ABB RobotStudio station: PROYECTO_BUENO_ROBOTICA.rspag

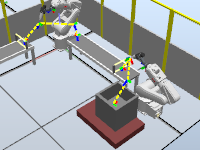
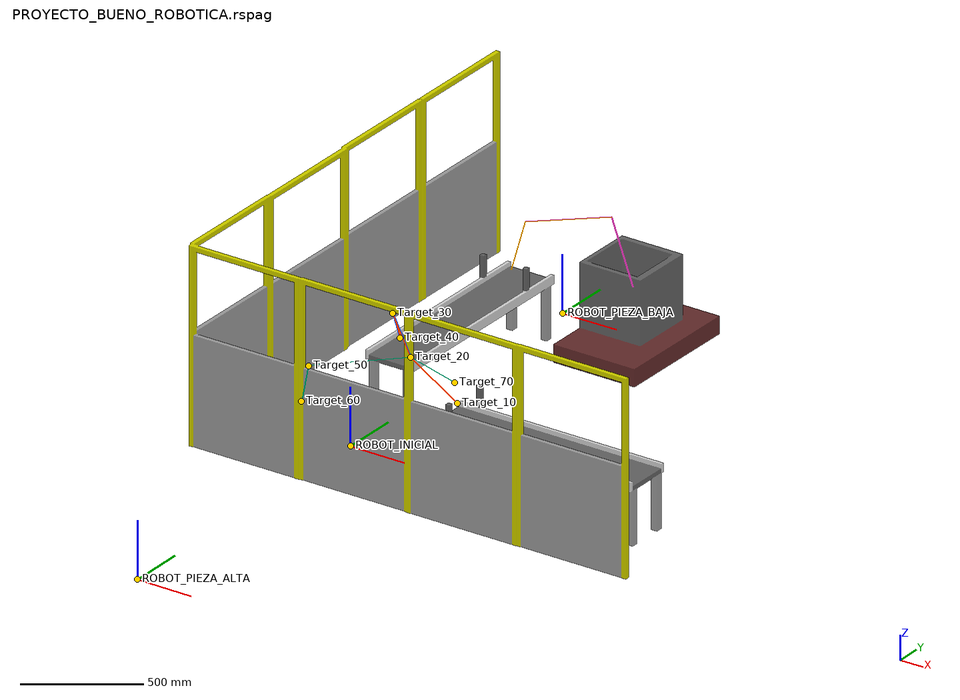
[picture v1: parts stored in the station drawn from their meshes, with robot base, taught points and paths (robot models come from the ABB library and are not in the file)]
--- station ---
Station Station (saved by RobotStudio 21.2.9526.0)
Controller Controlador3, task T_ROB1: task frame (RAPID world) sits at (0, 1493.87, 0) mm, rotated rx 0 ry 0 rz -90 deg in the station
Controller Controlador2, task T_ROB1: task frame (RAPID world) sits at (0, -1501.35, 0) mm, rotated rx 0 ry 0 rz 90 deg in the station
Controller Controlador1
  mechanical unit ROB_1: ROBOT_INICIAL, 6 joints, base frame (0, 0, 0) mm
Controller Controlador2
  mechanical unit ROB_1: ROBOT_PIEZA_ALTA, 6 joints, base frame (0, 0, 0) mm
Controller Controlador3
  mechanical unit ROB_1: ROBOT_PIEZA_BAJA, 6 joints, base frame (0, 0, 0) mm
Layout (positions relative to the parent item):
  - ROBOT_INICIAL [mechanism, from Robots\IRB120_3_58_G_01.rslib] at (0, 0, 0) mm; joint values [0.0153, -0.9412, 0.5438, -0.013, 0.8103, 0.021] (rad or m)
  - CINTA_INICIAL [part] at (1649.16, 0.65, 0) mm, rotated rx 0 ry 0 rz 180 deg, size 1004.2 x 233.8 x 295.1 mm
  - CINTA_PIEZA_BAJA [part] at (-5.09, 92.92, 0) mm, rotated rx 0 ry 0 rz 90 deg, size 1004.2 x 233.8 x 295.1 mm
  - ROBOT_PIEZA_BAJA [mechanism, from Robots\IRB120_3_58_G_01.rslib] at (0, 1493.87, 0) mm, rotated rx 0 ry 0 rz -90 deg; joint values [0, -1.3872, 0.8613, 0, 0.5297, 0] (rad or m)
  - ROBOT_PIEZA_ALTA [mechanism, from Robots\IRB120_3_58_G_01.rslib] at (0, -1501.35, 0) mm, rotated rx 0 ry 0 rz 90 deg; joint values [0, 0, 0, 0, 0.5236, 0] (rad or m)
  - PALE [part] at (-690.19, -1706.89, 0) mm
  - PALE_2 [part] at (226.17, 1105.11, 0) mm, size 400 x 600 x 80 mm
  - PALE_3 [part] at (-668.39, 1113.38, 0) mm
  - PALE_4 [part] at (309.1, -1704.29, 0) mm
  - MyTool [mechanism, from Training Objects\myTool.rslib] at (99.08, 0.84, 601.52) mm, rotated rx 178.96 ry 66.34 rz 179.16 deg
  - MyTool_3 [mechanism, from Training Objects\myTool.rslib] at (0, 1461.27, 551.16) mm, rotated rx 180 ry 89.78 rz 90 deg
  - PROTECCION_7 [part] at (1838.39, -653.58, 0) mm, rotated rx 0 ry 0 rz 90 deg, size 22.3 x 539.4 x 900 mm
  - PROTECCION_8 [part] at (-248.35, 2040.22, 0) mm, rotated rx 0 ry 0 rz 180 deg, size 22.3 x 539.4 x 900 mm
  - SENSOR [part] at (550.47, 98.45, 290.03) mm, size 20 x 20 x 100 mm
  - SENSOR_3 [part] at (31.03, 1015.51, 0) mm
  - SENSOR_4 [part] at (31.03, 1015.51, 0) mm
  - SENSOR_5 [part] at (31.03, 1015.51, 0) mm
  - CINTA_PIEZA_ALTA [part] at (-8.5, -1442.97, 0) mm, rotated rx 0 ry 0 rz 90 deg
  - SENSOR_6 [part] at (-130.12, -1151.13, 289.91) mm
  - SENSOR_7 [part] at (552.16, -120.97, 291.11) mm, size 20 x 20 x 100 mm
  - LineSensor_CINTA_INICIAL_ALTO [smart component, from Components\LineSensor.rslib]
      properties: Start=[0.562162 -0.10097 0.391108]; End=[0.560466 0.098451 0.39003]; Radius=0; SensedPart=SENSOR_7; SensedPoint=[0.562161987304687 -0.100970001220703 0.391108001708984]
    - _sensorPart_ [part], size 1.7 x 199.4 x 1.1 mm
  - LineSensor_CINTA_INICIAL_BAJO [smart component, from Components\LineSensor.rslib]
      properties: Start=[0.560466 0.098451 0.29003]; End=[0.562162 -0.10097 0.291108]; Radius=0; SensedPart=(none); SensedPoint=[0 0 0]
    - _sensorPart_ [part], size 1.7 x 199.4 x 1.1 mm
  - PhysicsControl [smart component, from Components\PhysicsControl.rslib]
      properties: Object=CINTA_INICIAL; Behavior=1; SurfaceVelocity=0.2
  - PhysicsControl_2 [smart component, from Components\PhysicsControl.rslib]
      properties: Object=CINTA_PIEZA_BAJA; Behavior=1; SurfaceVelocity=0.2
  - Attacher [smart component, from Components\Attacher.rslib]
      properties: Parent=MyTool; Flange=0; Child=(none); Mount=false; Offset=[0 0 0]; Orientation=[0 0 0]
  - Detacher [smart component, from Components\Detacher.rslib]
      properties: Child=(none); KeepPosition=true
  - SENSOR_8 [part] at (87, 1086.5, 290.62) mm, size 20 x 20 x 100 mm
  - SENSOR_9 [part] at (-126.77, 1089.55, 289.95) mm, size 20 x 20 x 100 mm
  - SENSOR_10 [part] at (89.27, -1145.05, 289.5) mm
  - LineSensor_CINTA:PIEZA_BAJA_ALTO [smart component, from Components\LineSensor.rslib]
      properties: Start=[0.085996 1.096498 0.390618]; End=[-0.099773 1.099547 0.389951]; Radius=0; SensedPart=(none); SensedPoint=[0 0 0]
    - _sensorPart_ [part], size 185.8 x 3 x 0.7 mm
  - LineSensor_CINTA_PIEZA_BAJA_BAJO [smart component, from Components\LineSensor.rslib]
      properties: Start=[0.076996 1.096498 0.290618]; End=[-0.098773 1.099547 0.289951]; Radius=0; SensedPart=(none); SensedPoint=[0 0 0]
    - _sensorPart_ [part], size 175.8 x 3 x 0.7 mm
  - CAJA [part] at (1364.14, -37.71, 266.99) mm, size 60 x 60 x 60 mm
  - Source [smart component, from Components\Source.rslib]
      properties: Source=CAJA; Copy=(none); Parent=(none); Position=[1.348944 -0.035764 0.27]; Orientation=[0 0 0]; Transient=true; PhysicsBehavior=3
  - Attacher_2 [smart component, from Components\Attacher.rslib]
      properties: Parent=MyTool_3; Flange=0; Child=(none); Mount=false; Offset=[0 0 0]; Orientation=[0 0 0]
  - Detacher_2 [smart component, from Components\Detacher.rslib]
      properties: Child=(none); KeepPosition=true
  - CAJA_GRANDE [part] at (1304.51, -24.93, 274) mm, size 100 x 100 x 150 mm
  - CAJA_GUARDAR [part] at (-496.56, 737.11, 75.2) mm, size 304.8 x 304.8 x 304.8 mm
  - PROTECCION_9 [part] at (225.18, -657.22, 0) mm, rotated rx 0 ry 0 rz 90 deg, size 22.3 x 539.4 x 900 mm
  - PROTECCION_10 [part] at (-242.45, 415.11, 0) mm, rotated rx 0 ry 0 rz 180 deg, size 22.3 x 539.4 x 900 mm
  - PROTECCION_11 [part] at (-239.98, 952.89, 0) mm, rotated rx 0 ry 0 rz 180 deg, size 22.3 x 539.4 x 900 mm
  - PROTECCION_12 [part] at (-248.62, 1492.56, 0) mm, rotated rx 0 ry 0 rz 180 deg, size 22.3 x 539.4 x 900 mm
  - PROTECCION_13 [part] at (764.68, -653.95, 0) mm, rotated rx 0 ry 0 rz 90 deg, size 22.3 x 539.4 x 900 mm
  - PROTECCION_14 [part] at (1298.16, -656.54, 0) mm, rotated rx 0 ry 0 rz 90 deg, size 22.3 x 539.4 x 900 mm
  - Sink [smart component, from Components\Sink.rslib]
      properties: Object=(none)
Attachment: MyTool is attached to ROBOT_INICIAL / Link6
Attachment: MyTool_3 is attached to ROBOT_PIEZA_BAJA / Link6
Station signals: DI CAJA
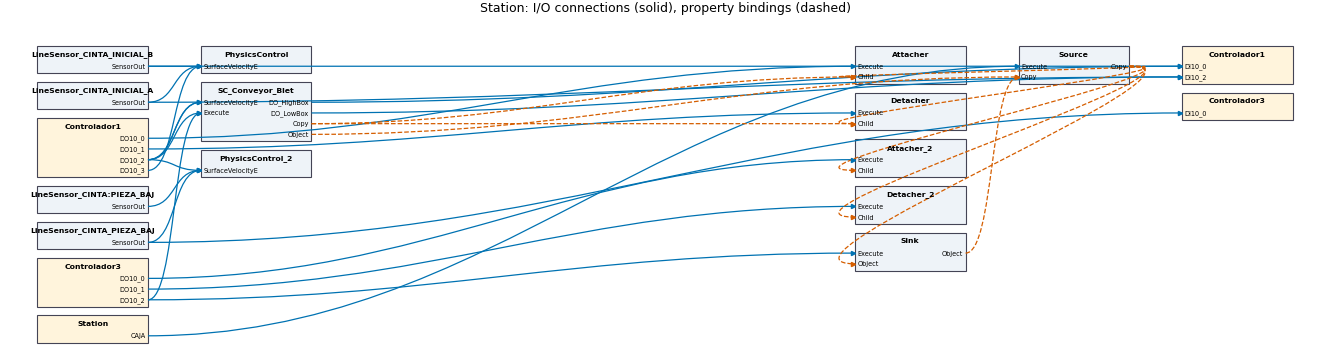
Station logic (signal -> signal, property => property):
  SC_Conveyor_Blet.DO_HighBox -> Controlador1.DI10_0
  SC_Conveyor_Blet.DO_LowBox -> Controlador1.DI10_2
  LineSensor_CINTA_INICIAL_BAJO.SensorOut -> PhysicsControl.SurfaceVelocityEnabled
  LineSensor_CINTA_INICIAL_ALTO.SensorOut -> PhysicsControl.SurfaceVelocityEnabled
  Controlador1.DO10_0 -> Attacher.Execute
  LineSensor_CINTA_INICIAL_BAJO.SensorOut -> Controlador1.DI10_0
  LineSensor_CINTA_INICIAL_ALTO.SensorOut -> Controlador1.DI10_2
  Controlador1.DO10_1 -> Detacher.Execute
  LineSensor_CINTA:PIEZA_BAJA_ALTO.SensorOut -> PhysicsControl_2.SurfaceVelocityEnabled
  LineSensor_CINTA_PIEZA_BAJA_BAJO.SensorOut -> PhysicsControl_2.SurfaceVelocityEnabled
  Controlador1.DO10_2 -> PhysicsControl_3.SurfaceVelocityEnabled
  Controlador1.DO10_3 -> PhysicsControl.SurfaceVelocityEnabled
  Controlador1.DO10_2 -> PhysicsControl_5.SurfaceVelocityEnabled
  Controlador1.DO10_2 -> Source.Execute
  Controlador1.DO10_2 -> PhysicsControl_2.SurfaceVelocityEnabled
  LineSensor_CINTA_PIEZA_BAJA_BAJO.SensorOut -> Controlador3.DI10_0
  Controlador3.DO10_0 -> Attacher_2.Execute
  Controlador3.DO10_1 -> Detacher_2.Execute
  Controlador3.DO10_2 -> Sink.Execute
  Controlador3.DO10_2 -> Sink.Execute
  Station.CAJA -> Source.Execute
  Source.Copy => Attacher.Child
  Source.Copy => Detacher.Child
  Source.Copy => Attacher.Child
  Source.Copy => Detacher.Child
  Source.Copy => Attacher_2.Child
  Source.Copy => Detacher_2.Child
  Sink.Object => Source.Copy
  Sink.Object => Source.Copy
  Source.Copy => Sink.Object

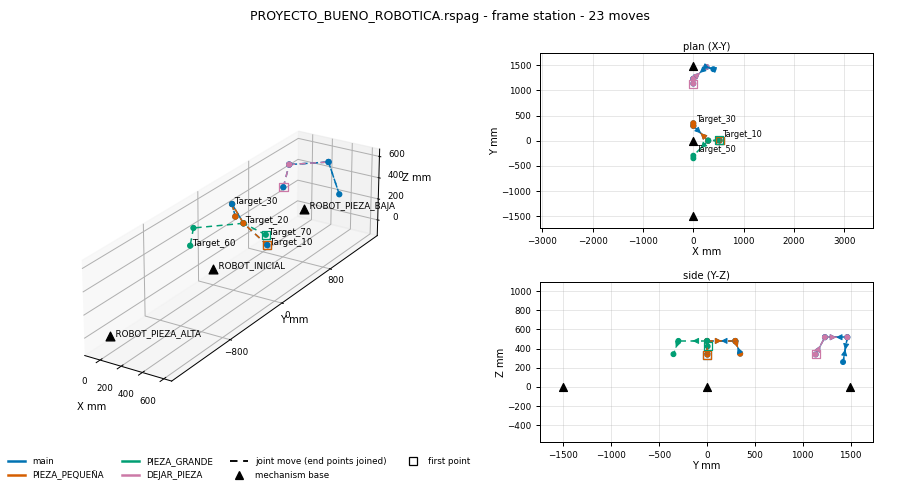
[picture p0: tool path of PROYECTO_BUENO_ROBOTICA.rspag in frame station, 23 of 23 moves have a stored position in this frame; points joined in program order, loops and branches not executed]
--- Backups/Controlador1/RAPID/TASK1/PROGMOD/CalibData.mod ---
MODULE CalibData
    PERS tooldata MyTool:=[TRUE,[[31.7926,0,229.639],[0.945519,0,0.325568,0]],[1,[0,0,1],[1,0,0,0],0,0,0]];
    TASK PERS wobjdata CINTA_1:=[FALSE,TRUE,"",[[0,0,0],[1,0,0,0]],[[0,0,0],[1,0,0,0]]];
ENDMODULE

--- Backups/Controlador1/RAPID/TASK1/PROGMOD/Module1.mod ---
MODULE Module1
        CONST robtarget Target_10:=[[524.488,5.564,337.068],[0.000000001,-0.000000001,1,0],[0,0,0,0],[9E+09,9E+09,9E+09,9E+09,9E+09,9E+09]];
    CONST robtarget Target_20:=[[296.669421919,2.08003687,480.265402411],[0.244840724,-0.000000001,0.969556084,0.003744278],[0,-1,0,0],[9E+09,9E+09,9E+09,9E+09,9E+09,9E+09]];
    CONST robtarget Target_30:=[[0.854294307,296.675483713,480.265402411],[0.171348121,-0.682180871,0.688961725,0.174930904],[1,-1,0,0],[9E+09,9E+09,9E+09,9E+09,9E+09,9E+09]];
    CONST robtarget Target_40:=[[0.578072629,347.819693408,346.913289479],[0.030324355,-0.70294026,0.709927462,0.03095842],[1,-1,0,0],[9E+09,9E+09,9E+09,9E+09,9E+09,9E+09]];
    CONST robtarget Target_50:=[[0.892731255,-296.675394938,480.265369004],[0.175434591,0.686950192,0.684206456,-0.170832265],[-1,-1,0,0],[9E+09,9E+09,9E+09,9E+09,9E+09,9E+09]];
    CONST robtarget Target_60:=[[1.479554637,-348.653016996,341.544953495],[0.025529615,0.708070337,0.705242245,-0.024859873],[-1,-1,0,0],[9E+09,9E+09,9E+09,9E+09,9E+09,9E+09]];
    CONST robtarget Target_70:=[[507.935,8.772,423.995],[0.000000001,-0.000000001,1,0],[0,0,0,0],[9E+09,9E+09,9E+09,9E+09,9E+09,9E+09]];
!***********************************************************
    !
    ! Módulo:  Module1
    !
    ! Descripción:
    !   <Introduzca la descripción aquí>
    !
    ! Autor: javie
    !
    ! Versión: 1.0
    !
    !***********************************************************


    !***********************************************************
    !
    ! Procedimiento Main
    !
    !   Este es el punto de entrada de su programa
    !
    !***********************************************************
    PROC main()
        Set DO10_4;
        Reset DO10_4;
        Set DO10_3;
        Reset DO10_1;
        Reset DO10_0;
        WaitDI DI10_0,1;
        WaitTime 1;
        MoveJ Target_10,v1000,fine,MyTool\WObj:=CINTA_1;
        Set DO10_0;
        WaitTime 1;
        MoveJ Target_20,v1000,fine,MyTool\WObj:=CINTA_1;
        Set DO10_4;
        MoveJ Target_30,v1000,z100,MyTool\WObj:=CINTA_1;
        MoveJ Target_40,v1000,fine,MyTool\WObj:=CINTA_1;
        Set DO10_1;
        Set DO10_2;
        WaitTime 1;
        MoveJ Target_30,v1000,z100,MyTool\WObj:=CINTA_1;
        MoveJ Target_20,v1000,fine,MyTool\WObj:=CINTA_1;


    ENDPROC
    PROC PIEZA_PEQUEÑA()
        MoveJ Target_10,v1000,fine,MyTool\WObj:=CINTA_1;
        MoveJ Target_20,v1000,fine,MyTool\WObj:=CINTA_1;
        MoveJ Target_30,v1000,z100,MyTool\WObj:=CINTA_1;
        MoveJ Target_40,v1000,fine,MyTool\WObj:=CINTA_1;
    ENDPROC
    PROC PIEZA_GRANDE()
        MoveJ Target_70,v200,fine,MyTool\WObj:=CINTA_1;
        MoveJ Target_20,v1000,fine,MyTool\WObj:=CINTA_1;
        MoveJ Target_50,v1000,fine,MyTool\WObj:=CINTA_1;
        MoveJ Target_60,v1000,fine,MyTool\WObj:=CINTA_1;
    ENDPROC
ENDMODULE

--- Backups/Controlador2/RAPID/TASK1/PROGMOD/Module1.mod ---
MODULE Module1
    !***********************************************************
    !
    ! Módulo:  Module1
    !
    ! Descripción:
    !   <Introduzca la descripción aquí>
    !
    ! Autor: javie
    !
    ! Versión: 1.0
    !
    !***********************************************************


    !***********************************************************
    !
    ! Procedimiento Main
    !
    !   Este es el punto de entrada de su programa
    !
    !***********************************************************
    PROC main()
        !Añada aquí su código
    ENDPROC
ENDMODULE

--- Backups/Controlador3/RAPID/TASK1/PROGMOD/CalibData.mod ---
MODULE CalibData
    PERS tooldata MyTool:=[TRUE,[[31.792631019,0,229.638935148],[0.945518576,0,0.325568154,0]],[1,[0,0,1],[1,0,0,0],0,0,0]];
ENDMODULE

--- Backups/Controlador3/RAPID/TASK1/PROGMOD/Module1.mod ---
MODULE Module1
        CONST robtarget Target_10:=[[358.458066847,0,338.786730568],[0.146240119,0,0.989249123,0],[0,0,0,0],[9E+09,9E+09,9E+09,9E+09,9E+09,9E+09]];
    CONST robtarget Target_20:=[[262.109517355,0,518.483225276],[0.43664348,0,0.899634632,0],[0,0,0,4],[9E+09,9E+09,9E+09,9E+09,9E+09,9E+09]];
    CONST robtarget Target_30:=[[28.317745802,260.57533337,518.483225276],[0.325004428,-0.600792335,0.669620072,0.291598441],[0,0,-1,4],[9E+09,9E+09,9E+09,9E+09,9E+09,9E+09]];
    CONST robtarget Target_40:=[[72.897632969,399.258136435,259.476555382],[0.009818398,-0.640410998,0.767925978,0.008188042],[0,0,-1,0],[9E+09,9E+09,9E+09,9E+09,9E+09,9E+09]];
    CONST robtarget Target_50:=[[124.528656109,351.162,140.028],[0,-0.707106781,0.707106782,0],[0,0,0,0],[9E+09,9E+09,9E+09,9E+09,9E+09,9E+09]];

!***********************************************************
    !
    ! Módulo:  Module1
    !
    ! Descripción:
    !   <Introduzca la descripción aquí>
    !
    ! Autor: javie
    !
    ! Versión: 1.0
    !
    !***********************************************************


    !***********************************************************
    !
    ! Procedimiento Main
    !
    !   Este es el punto de entrada de su programa
    !
    !***********************************************************
    PROC main()

       Reset DO10_0;
       Reset DO10_1;
       Reset DO10_2;
       WaitDI DI10_0,1;
       MoveJ Target_10,v200,fine,MyTool\WObj:=wobj0;
       WaitTime 1;
       Set DO10_0;
       WaitTime 0.5;
       MoveJ Target_20,v200,fine,MyTool\WObj:=wobj0;
       MoveJ Target_30,v200,fine,MyTool\WObj:=wobj0;
       MoveJ Target_40,v1000,z100,MyTool\WObj:=wobj0;
       Waittime 1;
       Set DO10_1;
       Set DO10_2;
       MoveJ Target_30,v200,fine,MyTool\WObj:=wobj0;
       MoveJ Target_20,v200,fine,MyTool\WObj:=wobj0;
       Set DO10_3;

    ENDPROC
    PROC DEJAR_PIEZA()
        MoveJ Target_10,v200,fine,MyTool\WObj:=wobj0;
        MoveJ Target_20,v1000,fine,MyTool\WObj:=wobj0;
        MoveJ Target_30,v1000,fine,MyTool\WObj:=wobj0;




    ENDPROC
ENDMODULE

--- Backups/Controlador1/SYSPAR/EIO.cfg ---
EIO:CFG_1.0:6:1::
#
INDUSTRIAL_NETWORK:

      -Name "DeviceNet" -Label "DeviceNet Master/Slave Network" -Address "2"
#
DEVICENET_DEVICE:

      -Name "d652" -VendorName "ABB Robotics" -ProductName "24 VDC I/O Device"\
      -Label "DSQC 652 24 VDC I/O Device" -Address 10 -ProductCode 26\
      -DeviceType 7 -ConnectionType "COS" -OutputSize 2 -InputSize 2
#
DEVICENET_INTERNAL_DEVICE:

      -Name "DN_Internal_Device" -VendorName "ABB Robotics"\
      -ProductName "DeviceNet Internal Slave Device"
#
EIO_SIGNAL:

      -Name "DI10_0" -SignalType "DI" -Device "d652" -DeviceMap "0"

      -Name "DI10_1" -SignalType "DI" -Device "d652" -DeviceMap "1"

      -Name "DI10_2" -SignalType "DI" -Device "d652" -DeviceMap "2"

      -Name "DI10_3" -SignalType "DI" -Device "d652" -DeviceMap "3"

      -Name "DO10_0" -SignalType "DO" -Device "d652" -DeviceMap "0"

      -Name "DO10_1" -SignalType "DO" -Device "d652" -DeviceMap "1"

      -Name "DO10_2" -SignalType "DO" -Device "d652" -DeviceMap "2"

      -Name "DO10_3" -SignalType "DO" -Device "d652" -DeviceMap "3"

      -Name "DO10_4" -SignalType "DO" -Device "d652" -DeviceMap "4"

--- Backups/Controlador3/SYSPAR/EIO.cfg ---
EIO:CFG_1.0:6:1::
#
INDUSTRIAL_NETWORK:

      -Name "DeviceNet" -Label "DeviceNet Master/Slave Network" -Address "2"
#
DEVICENET_DEVICE:

      -Name "d652" -VendorName "ABB Robotics" -ProductName "24 VDC I/O Device"\
      -Label "DSQC 652 24 VDC I/O Device" -Address 10 -ProductCode 26\
      -DeviceType 7 -ConnectionType "COS" -OutputSize 2 -InputSize 2
#
DEVICENET_INTERNAL_DEVICE:

      -Name "DN_Internal_Device" -VendorName "ABB Robotics"\
      -ProductName "DeviceNet Internal Slave Device"
#
EIO_SIGNAL:

      -Name "DI10_0" -SignalType "DI" -Device "d652" -DeviceMap "0"

      -Name "DI10_1" -SignalType "DI" -Device "d652" -DeviceMap "1"

      -Name "DI10_2" -SignalType "DI" -Device "d652" -DeviceMap "2"

      -Name "DO10_0" -SignalType "DO" -Device "d652" -DeviceMap "0"

      -Name "DO10_1" -SignalType "DO" -Device "d652" -DeviceMap "1"

      -Name "DO10_2" -SignalType "DO" -Device "d652" -DeviceMap "2"

      -Name "DO10_3" -SignalType "DO" -Device "d652" -DeviceMap "3"

      -Name "DO10_4" -SignalType "DO" -Device "d652" -DeviceMap "4"
